// TIA Portal V21 export
VAR_GLOBAL   // PLC tag table "K_Sequenza"
END_VAR
VAR_GLOBAL CONSTANT   // user constants
   K_Sequenza_Lavaggio : Int := 1;   // Washing / Lavaggio
   K_Sequenza_Produzione : Int := 2;   // Produktion / Production / Producción / Produzione
END_VAR
